// TwinCAT 3 PLC project SimPLC
// ProgramVersion: 3.1.4023.0
// libraries:
//   Tc2_EtherCAT, * (Beckhoff Automation GmbH)
//   Tc2_Standard, * (Beckhoff Automation GmbH)
//   Tc2_System, * (Beckhoff Automation GmbH)
//   Tc2_Utilities, * (Beckhoff Automation GmbH)
//   Tc3_Module, * (Beckhoff Automation GmbH)
// project tree:
//   DUTs/ ST_EC_SIM_Device_Inputs.TcDUT
//   / PlcTask.TcTTO
//   POUs/ FB_EL4102_Sim.TcPOU, MAIN.TcPOU, PRG_AnalogSim.TcPOU, PRG_EncoderSim.TcPOU, PRG_EtherCATSimMasterDiag.TcPOU, PRG_SystemFunctions.TcPOU
// real-time tasks:
//   TASK PlcTask: cycle T#62.5us, priority 6, ADS port 350
// I/O:
//   DEVICE EtherCAT Simulation 1, AmsNetId 5.62.33.82.2.1
//     Term 1 (EK1100) // EK1100-0000-0018
//     Term 2 (EL5001) // EL5001-0000-1021
//     Term 4 (EL4102) // EL4102-0000-1020
//   DEVICE EtherCAT Simulation 2, AmsNetId 5.62.33.82.3.1
//     Term 1 (EK1100) // EK1100-0000-0018
//     Term 2 (EL5001) // EL5001-0000-1021
//     Term 4 (EL4102) // EL4102-0000-1020
//   DEVICE EtherCAT Simulation 3, AmsNetId 5.62.33.82.4.1
//     Term 1 (EK1100) // EK1100-0000-0018
//     Term 2 (EL5001) // EL5001-0000-1021
//     Term 4 (EL4102) // EL4102-0000-1020
//   DEVICE EtherCAT Simulation 4, AmsNetId 5.62.33.82.5.1
//     Term 1 (EK1100) // EK1100-0000-0018
//     Term 2 (EL5001) // EL5001-0000-1021
//     Term 4 (EL4102) // EL4102-0000-1020
//   DEVICE EtherCAT Simulation 5, AmsNetId 5.62.33.82.6.1
//     Term 1 (EK1100) // EK1100-0000-0018
//     Term 2 (EL5001) // EL5001-0000-1021
//     Term 4 (EL4102) // EL4102-0000-1020
//   DEVICE EtherCAT Simulation 6, AmsNetId 5.62.33.82.7.1
//     Term 1 (EK1100) // EK1100-0000-0018
//     Term 2 (EL5001) // EL5001-0000-1021
//     Term 4 (EL4102) // EL4102-0000-1020
//   DEVICE Local (EtherCAT), AmsNetId 5.24.131.22.11.1
//     Term 1 (EK1200) [EK1200-5000 EtherCAT Power supply (2A E-Bus)]
//       Term 2 (EL6070) [EL6070 1Ch. Licensing-Terminal]
//       Term 3 (EL9011) [EL9011 End Terminal]
// variable links:
//   SimPLC Instance <-> EtherCAT Simulation 1
//     PlcTask Inputs/PRG_EtherCATSimMasterDiag.EcSimNetorkDiag[1]/AmsNetId <-> Inputs/AmsNetId
//     PlcTask Inputs/PRG_EtherCATSimMasterDiag.EcSimNetorkDiag[1]/Dc_Time <-> Inputs/Dc Time
//     PlcTask Inputs/PRG_EtherCATSimMasterDiag.EcSimNetorkDiag[1]/Dc_Time_to_System_Time_Offset <-> Inputs/Dc Time to System Time Offset
//     PlcTask Inputs/PRG_EtherCATSimMasterDiag.EcSimNetorkDiag[1]/DevState <-> Inputs/DevState
//     PlcTask Inputs/PRG_EtherCATSimMasterDiag.EcSimNetorkDiag[1]/Status <-> Inputs/Status
//     PlcTask Inputs/PRG_EtherCATSimMasterDiag.EcSimNetorkDiag[1]/Telegram_Counter <-> Inputs/Telegram Counter
//   SimPLC Instance <-> EtherCAT Simulation 1/Term 2 (EL5001)
//     PlcTask Outputs/PRG_EncoderSim.SimEncoderCount <-> SSI Inputs/Counter value
//   SimPLC Instance <-> EtherCAT Simulation 1/Term 4 (EL4102)
//     PlcTask Inputs/PRG_AnalogSim.arEL4102[1].Ch1 <-> Channel 1/Output
//     PlcTask Inputs/PRG_AnalogSim.arEL4102[1].Ch2 <-> Channel 2/Output
//   SimPLC Instance <-> EtherCAT Simulation 2
//     PlcTask Inputs/PRG_EtherCATSimMasterDiag.EcSimNetorkDiag[2]/AmsNetId <-> Inputs/AmsNetId
//     PlcTask Inputs/PRG_EtherCATSimMasterDiag.EcSimNetorkDiag[2]/Dc_Time <-> Inputs/Dc Time
//     PlcTask Inputs/PRG_EtherCATSimMasterDiag.EcSimNetorkDiag[2]/Dc_Time_to_System_Time_Offset <-> Inputs/Dc Time to System Time Offset
//     PlcTask Inputs/PRG_EtherCATSimMasterDiag.EcSimNetorkDiag[2]/DevState <-> Inputs/DevState
//     PlcTask Inputs/PRG_EtherCATSimMasterDiag.EcSimNetorkDiag[2]/Status <-> Inputs/Status
//     PlcTask Inputs/PRG_EtherCATSimMasterDiag.EcSimNetorkDiag[2]/Telegram_Counter <-> Inputs/Telegram Counter
//   SimPLC Instance <-> EtherCAT Simulation 2/Term 2 (EL5001)
//     PlcTask Outputs/PRG_EncoderSim.SimEncoderCount <-> SSI Inputs/Counter value
//   SimPLC Instance <-> EtherCAT Simulation 2/Term 4 (EL4102)
//     PlcTask Inputs/PRG_AnalogSim.arEL4102[2].Ch1 <-> Channel 1/Output
//     PlcTask Inputs/PRG_AnalogSim.arEL4102[2].Ch2 <-> Channel 2/Output
//   SimPLC Instance <-> EtherCAT Simulation 3
//     PlcTask Inputs/PRG_EtherCATSimMasterDiag.EcSimNetorkDiag[3]/AmsNetId <-> Inputs/AmsNetId
//     PlcTask Inputs/PRG_EtherCATSimMasterDiag.EcSimNetorkDiag[3]/Dc_Time <-> Inputs/Dc Time
//     PlcTask Inputs/PRG_EtherCATSimMasterDiag.EcSimNetorkDiag[3]/Dc_Time_to_System_Time_Offset <-> Inputs/Dc Time to System Time Offset
//     PlcTask Inputs/PRG_EtherCATSimMasterDiag.EcSimNetorkDiag[3]/DevState <-> Inputs/DevState
//     PlcTask Inputs/PRG_EtherCATSimMasterDiag.EcSimNetorkDiag[3]/Status <-> Inputs/Status
//     PlcTask Inputs/PRG_EtherCATSimMasterDiag.EcSimNetorkDiag[3]/Telegram_Counter <-> Inputs/Telegram Counter
//   SimPLC Instance <-> EtherCAT Simulation 3/Term 2 (EL5001)
//     PlcTask Outputs/PRG_EncoderSim.SimEncoderCount <-> SSI Inputs/Counter value
//   SimPLC Instance <-> EtherCAT Simulation 3/Term 4 (EL4102)
//     PlcTask Inputs/PRG_AnalogSim.arEL4102[3].Ch1 <-> Channel 1/Output
//     PlcTask Inputs/PRG_AnalogSim.arEL4102[3].Ch2 <-> Channel 2/Output
//   SimPLC Instance <-> EtherCAT Simulation 4
//     PlcTask Inputs/PRG_EtherCATSimMasterDiag.EcSimNetorkDiag[4]/AmsNetId <-> Inputs/AmsNetId
//     PlcTask Inputs/PRG_EtherCATSimMasterDiag.EcSimNetorkDiag[4]/Dc_Time <-> Inputs/Dc Time
//     PlcTask Inputs/PRG_EtherCATSimMasterDiag.EcSimNetorkDiag[4]/Dc_Time_to_System_Time_Offset <-> Inputs/Dc Time to System Time Offset
//     PlcTask Inputs/PRG_EtherCATSimMasterDiag.EcSimNetorkDiag[4]/DevState <-> Inputs/DevState
//     PlcTask Inputs/PRG_EtherCATSimMasterDiag.EcSimNetorkDiag[4]/Status <-> Inputs/Status
//     PlcTask Inputs/PRG_EtherCATSimMasterDiag.EcSimNetorkDiag[4]/Telegram_Counter <-> Inputs/Telegram Counter
//   SimPLC Instance <-> EtherCAT Simulation 4/Term 2 (EL5001)
//     PlcTask Outputs/PRG_EncoderSim.SimEncoderCount <-> SSI Inputs/Counter value
//   SimPLC Instance <-> EtherCAT Simulation 4/Term 4 (EL4102)
//     PlcTask Inputs/PRG_AnalogSim.arEL4102[4].Ch1 <-> Channel 1/Output
//     PlcTask Inputs/PRG_AnalogSim.arEL4102[4].Ch2 <-> Channel 2/Output
//   SimPLC Instance <-> EtherCAT Simulation 5
//     PlcTask Inputs/PRG_EtherCATSimMasterDiag.EcSimNetorkDiag[5]/AmsNetId <-> Inputs/AmsNetId
//     PlcTask Inputs/PRG_EtherCATSimMasterDiag.EcSimNetorkDiag[5]/Dc_Time <-> Inputs/Dc Time
//     PlcTask Inputs/PRG_EtherCATSimMasterDiag.EcSimNetorkDiag[5]/Dc_Time_to_System_Time_Offset <-> Inputs/Dc Time to System Time Offset
//     PlcTask Inputs/PRG_EtherCATSimMasterDiag.EcSimNetorkDiag[5]/DevState <-> Inputs/DevState
//     PlcTask Inputs/PRG_EtherCATSimMasterDiag.EcSimNetorkDiag[5]/Status <-> Inputs/Status
//     PlcTask Inputs/PRG_EtherCATSimMasterDiag.EcSimNetorkDiag[5]/Telegram_Counter <-> Inputs/Telegram Counter
//   SimPLC Instance <-> EtherCAT Simulation 5/Term 2 (EL5001)
//     PlcTask Outputs/PRG_EncoderSim.SimEncoderCount <-> SSI Inputs/Counter value
//   SimPLC Instance <-> EtherCAT Simulation 5/Term 4 (EL4102)
//     PlcTask Inputs/PRG_AnalogSim.arEL4102[5].Ch1 <-> Channel 1/Output
//     PlcTask Inputs/PRG_AnalogSim.arEL4102[5].Ch2 <-> Channel 2/Output
//   SimPLC Instance <-> EtherCAT Simulation 6
//     PlcTask Inputs/PRG_EtherCATSimMasterDiag.EcSimNetorkDiag[6]/AmsNetId <-> Inputs/AmsNetId
//     PlcTask Inputs/PRG_EtherCATSimMasterDiag.EcSimNetorkDiag[6]/Dc_Time <-> Inputs/Dc Time
//     PlcTask Inputs/PRG_EtherCATSimMasterDiag.EcSimNetorkDiag[6]/Dc_Time_to_System_Time_Offset <-> Inputs/Dc Time to System Time Offset
//     PlcTask Inputs/PRG_EtherCATSimMasterDiag.EcSimNetorkDiag[6]/DevState <-> Inputs/DevState
//     PlcTask Inputs/PRG_EtherCATSimMasterDiag.EcSimNetorkDiag[6]/Status <-> Inputs/Status
//     PlcTask Inputs/PRG_EtherCATSimMasterDiag.EcSimNetorkDiag[6]/Telegram_Counter <-> Inputs/Telegram Counter
//   SimPLC Instance <-> EtherCAT Simulation 6/Term 2 (EL5001)
//     PlcTask Outputs/PRG_EncoderSim.SimEncoderCount <-> SSI Inputs/Counter value
//   SimPLC Instance <-> EtherCAT Simulation 6/Term 4 (EL4102)
//     PlcTask Inputs/PRG_AnalogSim.arEL4102[6].Ch1 <-> Channel 1/Output
//     PlcTask Inputs/PRG_AnalogSim.arEL4102[6].Ch2 <-> Channel 2/Output
//   SimPLC Instance <-> Local (EtherCAT)
//     PlcTask Inputs/MAIN.LocalEtherCATDevState <-> Inputs/DevState

CONFIGURATION SimPLC
    RESOURCE PLC ON TwinCAT3
        TASK PlcTask(INTERVAL := T#62.5us, PRIORITY := 6);
        PROGRAM MAIN WITH PlcTask : MAIN;
    END_RESOURCE
END_CONFIGURATION

// ---- DUTs/ST_EC_SIM_Device_Inputs.TcDUT
TYPE ST_EC_SIM_Device_Inputs :
STRUCT
	Status							:UDINT;
	Telegram_Counter				:UDINT;
	Dc_Time							:ULINT;
	Dc_Time_to_System_Time_Offset	:ULINT;
	{attribute 'displaymode':='hex'} 
	DevState						:UINT;
	AmsNetId						:AMSNETID;
END_STRUCT
END_TYPE

// ---- POUs/MAIN.TcPOU
{attribute 'TcCallAfterOutputUpdate'}
PROGRAM MAIN
VAR
	LocalEtherCATDevState	AT%I*:UINT ;
END_VAR

PRG_EtherCATSimMasterDiag();

PRG_EncoderSim();

PRG_AnalogSim();

PRG_SystemFunctions();

END_PROGRAM

// ---- POUs/PRG_EtherCATSimMasterDiag.TcPOU
PROGRAM PRG_EtherCATSimMasterDiag
VAR
	EcSimNetorkDiag		AT%I* 	:ARRAY[1..NumOfEcSimNetWorks] OF ST_EC_SIM_Device_Inputs;
	EcDevState					:ARRAY[1..NumOfEcSimNetWorks] OF STRING;
END_VAR
VAR CONSTANT
	NumOfEcSimNetWorks			:UDINT:=6;
END_VAR
VAR_TEMP
	i							:UDINT;
END_VAR


FOR i:=1 TO NumOfEcSimNetWorks DO
	EcDevState[i]:=F_ConvMasterDevStateToString(nState:=EcSimNetorkDiag[i].DevState);
END_FOR

END_PROGRAM

// ---- POUs/PRG_EncoderSim.TcPOU
PROGRAM PRG_EncoderSim
VAR
	SimEncoderCount	AT%Q*	:UDINT:=1;	
END_VAR

SimEncoderCount:=SimEncoderCount+1;

IF SimEncoderCount>=4096 THEN
	SimEncoderCount:=1;
END_IF

END_PROGRAM

// ---- POUs/PRG_AnalogSim.TcPOU
PROGRAM PRG_AnalogSim
VAR
	arEL4102			:ARRAY[1..NumOfEL4102] OF FB_EL4102_Sim;
END_VAR
VAR CONSTANT
	NumOfEL4102			:INT:=6;
END_VAR
VAR_TEMP
	i					:INT;
END_VAR

FOR i:=1 TO NumOfEL4102 DO
	arEL4102[i]();
END_FOR

END_PROGRAM

// ---- POUs/FB_EL4102_Sim.TcPOU
FUNCTION_BLOCK FB_EL4102_Sim
VAR_INPUT
END_VAR
VAR_OUTPUT
END_VAR
VAR
	Ch1				AT%I*	:INT;
	Ch2				AT%I*	:INT;	

	Ch1NotEqualToCh2		:UDINT;
	Delta					:INT;	
END_VAR

IF Ch1<>0 AND Ch2<>0 THEN
	IF Ch1 <> Ch2 THEN
		Delta				:=Ch1-Ch2;
		Ch1NotEqualToCh2	:=Ch1NotEqualToCh2+1;
	ELSE
		Delta:=0;
	END_IF
END_IF

END_FUNCTION_BLOCK

// ---- POUs/PRG_SystemFunctions.TcPOU
PROGRAM PRG_SystemFunctions
VAR
	xReboot			:BOOL;
	fbReboot		:NT_Reboot;
END_VAR

fbReboot(
	NETID:='' , 
	DELAY:=0, 
	START:=xReboot);

END_PROGRAM
